{attribute 'OPC.UA.DA.StructuredType' := '1'}
TYPE ST_GasMeterState :
STRUCT
	fVolume					: REAL;
	sVolumeUnit				: STRING := 'm3';
	fTemperature			: REAL;
	sTemperatureUnit		: STRING := 'degreeC';
	fVolumeFlowRate			: REAL;
	sVolumeFlowRateUnit		: STRING := 'm3/h';
END_STRUCT
END_TYPE

(* stored: Version 1.1.0.1, ProductVersion 3.1.4024.10
   DUT ST_GasMeterState: Id {8f2a4e18-73c7-4d66-a877-3aadfaffa2e2} *)
